// TIA Portal V17 export
// export: Created 2023-06-23T18:33:38.3691724Z, ExportSetting WithDefaults, DisplayName Totally Integrated Automation Portal, DisplayVersion V17, DisplayName TIA Portal Openness, DisplayVersion V17, DisplayName TIA Portal Version Control Interface, DisplayVersion V17, DisplayName STEP 7 Professional, DisplayVersion V17, DisplayName STEP 7 Safety, DisplayVersion V17, DisplayName WinCC Advanced / Unified PC, DisplayVersion V17
VAR_GLOBAL   // PLC tag table "09_CT-3"
   "iCT-3" AT %I8.0 : Bool;
   "oCT-3s" AT %Q20.6 : Bool;
   "oCT-3f" AT %Q20.7 : Bool;
END_VAR
